// TIA Portal V20 export
FUNCTION_BLOCK "Central_Auto_Control"   // FB21, LAD
{ S7_Optimized_Access := 'TRUE' }
// stored: MemoryReserve 100, SetENOAutomatically false
   VAR
      Auto_Turn_On : Bool;
      "Step" : Int;
      CS_Drive : Bool;
      SS_Go_H3 : Bool;
      SS_Go_H5 : Bool;
      SS_Go_CS : Bool;
      CS_Auto_Hyd_Up : Bool;
      CS_Auto_Hyd_Down : Bool;
      Step_Delay { S7_SetPoint := 'True'} : TON_TIME;
      Timer_active { S7_SetPoint := 'True'} : Bool;
   END_VAR
BEGIN

REGION Network 1
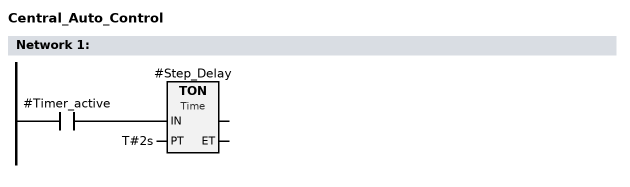
   RUNG wire#powerrail
      Contact( #Timer_active )
      { S7_Templates := "time_type := Time" } #Step_Delay.TON(pt := T#2s, et =>)
   END_RUNG
   // the same network as SCL:
   #Step_Delay(IN := #Timer_active, PT := T#2s);   // TON
END_REGION

REGION Network 2 (SCL)
   IF #Auto_Turn_On  AND "HMI_Central_Shifter".CS_Auto_Pos_Start <> 0  AND "HMI_Central_Shifter".CS_Auto_Pos_End <> 0  THEN
       IF #Step = 0 THEN  //drive CS to Start pos
           IF "CentralShifter_DB".CentralShifter_SideShifters_Instance.Hyd_Down_Status = 2 AND "CentralShifter_DB".CentralShifter_SideShifters_Instance.qLeftSide_in_Mid AND "CentralShifter_DB".CentralShifter_SideShifters_Instance.qRightSide_in_Mid AND NOT "iCS_SensorHoming_Left" AND NOT "iCS_SensorHoming_Right" THEN
               "HMI_Central_Shifter".CS_Destination_Pos := ("HMI_Central_Shifter".CS_Auto_Pos_Start MOD 10) + 6;
               #CS_Drive := 1;
           END_IF;
           IF "CentralShifter_DB".Arrived_Pos = ("HMI_Central_Shifter".CS_Auto_Pos_Start MOD 10) + 6 THEN
               #Timer_active := 1;
               IF #Step_Delay.Q THEN
                   #Step := 1;
                   #Timer_active := 0;
               END_IF;
           END_IF;

       ELSIF #Step = 1 THEN  //Drive SS to Start pos
           IF "CentralShifter_DB".Arrived_Pos <> ("HMI_Central_Shifter".CS_Auto_Pos_Start MOD 10) + 6 THEN
               #Timer_active := 1;
               IF #Step_Delay.Q THEN
                   #Step := 0;
                   #Timer_active := 0;
               END_IF;

           ELSIF "CentralShifter_DB".Arrived_Pos = ("HMI_Central_Shifter".CS_Auto_Pos_Start MOD 10) + 6 AND "CentralShifter_DB".CentralShifter_SideShifters_Instance.Hyd_Down_Status = 2 THEN
               IF "HMI_Central_Shifter".CS_Auto_Pos_Start < 10 THEN
                   #SS_Go_H5 := 1;
                   IF "CentralShifter_DB".CentralShifter_SideShifters_Instance.Sides_In_H5_Pos THEN
                       #Timer_active := 1;
                       IF #Step_Delay.Q THEN
                           #SS_Go_H5 := 0;
                           #Step := 2;
                           #Timer_active := 0;
                       END_IF;
                   END_IF;

               ELSIF "HMI_Central_Shifter".CS_Auto_Pos_Start > 10 THEN
                   #SS_Go_H3 := 1;
                   IF "CentralShifter_DB".CentralShifter_SideShifters_Instance.Sides_In_H3_Pos THEN
                       #Timer_active := 1;
                       IF #Step_Delay.Q THEN
                           #SS_Go_H3 := 0;
                           #Step := 2;
                           #Timer_active := 0;
                       END_IF;
                   END_IF;
               END_IF;
           END_IF;

       ELSIF #Step = 2 THEN  //Hyd UP SS on station
           IF NOT "CentralShifter_DB".CentralShifter_SideShifters_Instance.Sides_In_H3_Pos AND NOT "CentralShifter_DB".CentralShifter_SideShifters_Instance.Sides_In_H5_Pos AND "CentralShifter_DB".CentralShifter_SideShifters_Instance.Hyd_Down_Status = 2 THEN
               #Timer_active := 1;
               IF #Step_Delay.Q THEN
                   #Step := 1;
                   #Timer_active := 0;
               END_IF;
           ELSE
               #CS_Auto_Hyd_Up := 1;
           END_IF;
           IF "CentralShifter_DB".CentralShifter_SideShifters_Instance.Hyd_Up_Status = 2 THEN
               #CS_Auto_Hyd_Up := 0;
               #Timer_active := 1;
               IF #Step_Delay.Q THEN
                   #Step := 3;
                   #Timer_active := 0;
               END_IF;
           END_IF;

       ELSIF #Step = 3 THEN  //Drive SS to CS
           IF "CentralShifter_DB".CentralShifter_SideShifters_Instance.Hyd_Up_Status = 2 THEN
               #SS_Go_CS := 1;
               //ELSE
               //#Step := 2;
           END_IF;

           IF "CentralShifter_DB".CentralShifter_SideShifters_Instance.Sides_In_CS_Pos THEN
               #Timer_active := 1;
               IF #Step_Delay.Q THEN
                   #Step := 4;
                   #SS_Go_CS := 0;
                   #Timer_active := 0;
               END_IF;
           END_IF;

       ELSIF #Step = 4 THEN //hyd down on CS
           IF "CentralShifter_DB".CentralShifter_SideShifters_Instance.Sides_In_CS_Pos THEN
               #CS_Auto_Hyd_Down := 1;

               IF "CentralShifter_DB".CentralShifter_SideShifters_Instance.Hyd_Down_Status = 2 THEN
                   #Timer_active := 1;
                   IF #Step_Delay.Q THEN
                       #Step := 5;
                       #SS_Go_CS := 0;
                       #Timer_active := 0;
                   END_IF;
               END_IF;

           ELSE
               #SS_Go_CS := 1;
           END_IF;


       ELSIF #Step = 5 THEN //CS Drive 
           IF "CentralShifter_DB".CentralShifter_SideShifters_Instance.Hyd_Down_Status = 2 THEN
               "HMI_Central_Shifter".CS_Destination_Pos := ("HMI_Central_Shifter".CS_Auto_Pos_End MOD 10) + 6;
               #CS_Drive := 1;
           ELSE
               #Timer_active := 1;
               IF #Step_Delay.Q THEN
                   #Step := 4;
                   #Timer_active := 0;
               END_IF;
           END_IF;

           IF "CentralShifter_DB".Arrived_Pos = ("HMI_Central_Shifter".CS_Auto_Pos_End MOD 10) + 6 THEN
               #Timer_active := 1;
               IF #Step_Delay.Q THEN
                   #Step := 6;
                   #Timer_active := 0;
               END_IF;
           END_IF;

       ELSIF #Step = 6 THEN //Hyd Up on CS
           IF "CentralShifter_DB".CentralShifter_SideShifters_Instance.Sides_In_CS_Pos AND "CentralShifter_DB".Arrived_Pos = ("HMI_Central_Shifter".CS_Auto_Pos_End MOD 10) + 6 THEN
               #CS_Auto_Hyd_Up := 1;
               #SS_Go_CS := 0;
           ELSE
               #SS_Go_CS := 1;
           END_IF;
           IF "CentralShifter_DB".CentralShifter_SideShifters_Instance.Hyd_Up_Status = 2 THEN
               #Timer_active := 1;
               IF #Step_Delay.Q THEN
                   #CS_Auto_Hyd_Up := 0;
                   #SS_Go_CS := 0;
                   #Step := 7;
                   #Timer_active := 0;
               END_IF;
           END_IF;

       ELSIF #Step = 7 THEN //SS Drive to end pos
           IF "CentralShifter_DB".Arrived_Pos <> ("HMI_Central_Shifter".CS_Auto_Pos_End MOD 10) + 6 THEN
               #Timer_active := 1;
               IF #Step_Delay.Q THEN
                   #Step := 6;
                   #Timer_active := 0;
               END_IF;

           ELSIF "CentralShifter_DB".Arrived_Pos = ("HMI_Central_Shifter".CS_Auto_Pos_End MOD 10) + 6 THEN
               IF "HMI_Central_Shifter".CS_Auto_Pos_End < 10 THEN
                   #SS_Go_H5 := 1;
                   IF "CentralShifter_DB".CentralShifter_SideShifters_Instance.Sides_In_H5_Pos THEN
                       #Timer_active := 1;
                       IF #Step_Delay.Q THEN
                           #SS_Go_H5 := 0;
                           #Step := 8;
                           #Timer_active := 0;
                       END_IF;
                   END_IF;

               ELSIF "HMI_Central_Shifter".CS_Auto_Pos_End > 10 THEN
                   #SS_Go_H3 := 1;
                   IF "CentralShifter_DB".CentralShifter_SideShifters_Instance.Sides_In_H3_Pos THEN
                       #Timer_active := 1;
                       IF #Step_Delay.Q THEN
                           #SS_Go_H3 := 0;
                           #Step := 8;
                           #Timer_active := 0;
                       END_IF;
                   END_IF;
               END_IF;
           END_IF;

       ELSIF #Step = 8 THEN //Hyd down
           IF NOT "CentralShifter_DB".CentralShifter_SideShifters_Instance.Sides_In_H3_Pos AND NOT "CentralShifter_DB".CentralShifter_SideShifters_Instance.Sides_In_H5_Pos AND "CentralShifter_DB".CentralShifter_SideShifters_Instance.Hyd_Up_Status = 2 THEN
               #Timer_active := 1;
               IF #Step_Delay.Q THEN
                   #Step := 7;
                   #Timer_active := 0;
               END_IF;
           ELSE
               #CS_Auto_Hyd_Down := 1;
           END_IF;
           IF "CentralShifter_DB".CentralShifter_SideShifters_Instance.Hyd_Down_Status = 2 THEN
               #Timer_active := 1;
               IF #Step_Delay.Q THEN
                   #CS_Auto_Hyd_Down := 0;
                   #Step := 9;
                   #Timer_active := 0;
               END_IF;
           END_IF;

       ELSIF #Step = 9 THEN
           IF "CentralShifter_DB".CentralShifter_SideShifters_Instance.Hyd_Down_Status = 2 THEN
               #SS_Go_CS := 1;
           ELSE
               #Timer_active := 1;
               IF #Step_Delay.Q THEN
                   #Step := 8;
                   #Timer_active := 0;
               END_IF;
           END_IF;

           IF "CentralShifter_DB".CentralShifter_SideShifters_Instance.Sides_In_CS_Pos THEN
               #Timer_active := 1;
               IF #Step_Delay.Q THEN
                   #Step := 10;
                   #Timer_active := 0;
               END_IF;
           END_IF;
       END_IF;

   ELSE
       #CS_Drive := 0;
       #SS_Go_CS := 0;
       #SS_Go_H3 := 0;
       #SS_Go_H5 := 0;
       #CS_Auto_Hyd_Down := 0;
       #CS_Auto_Hyd_Up := 0;
       #Timer_active := 0;
       IF #Step = 10 THEN
           #Step := 0;
       END_IF;
   END_IF;
END_REGION
END_FUNCTION_BLOCK
